Xinje XDPPro project, PLC1: XD3-16 (software 3.7.17b 2023-10-13)

PROGRAM Ladder

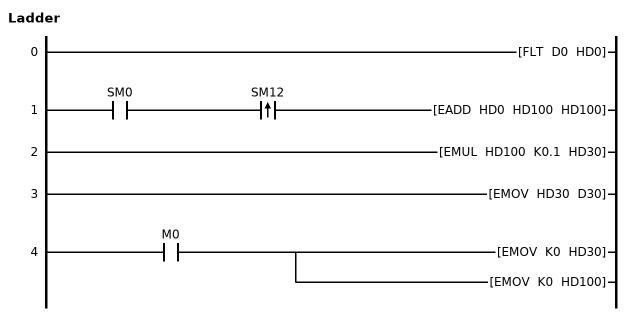
FLT    D0 HD0
LD     SM0
ANDP   SM12
EADD   HD0 HD100 HD100
EMUL   HD100 K0.1 HD30
EMOV   HD30 D30
LD     M0
EMOV   K0 HD30
EMOV   K0 HD100